PROGRAM Axis05_Auto
VAR
//System_Bit
	Always_ON	:	BOOL	:=TRUE	;//상시 ON 
	Always_OFF	:	BOOL	:=FALSE	;//상시 OFF
END_VAR

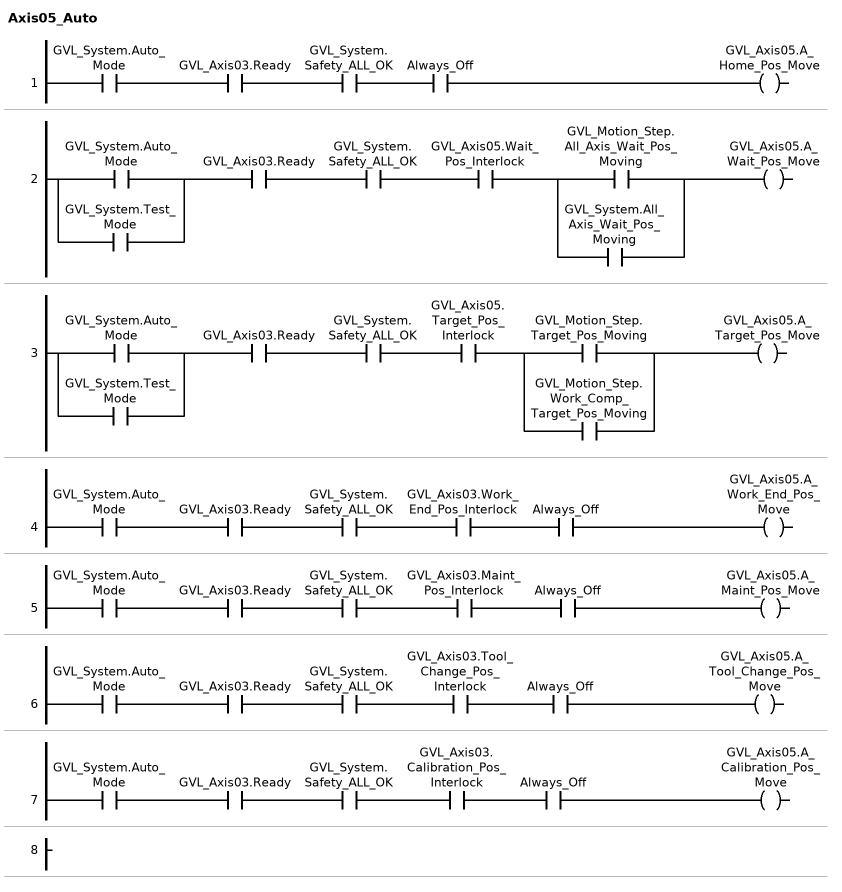
// NETWORK 1
GVL_Axis05.A_Home_Pos_Move := GVL_System.Auto_Mode AND GVL_Axis03.Ready AND GVL_System.Safety_ALL_OK AND Always_Off;

// NETWORK 2
GVL_Axis05.A_Wait_Pos_Move := (GVL_System.Auto_Mode OR GVL_System.Test_Mode) AND GVL_Axis03.Ready AND GVL_System.Safety_ALL_OK AND GVL_Axis05.Wait_Pos_Interlock AND (GVL_Motion_Step.All_Axis_Wait_Pos_Moving OR GVL_System.All_Axis_Wait_Pos_Moving);

// NETWORK 3
GVL_Axis05.A_Target_Pos_Move := (GVL_System.Auto_Mode OR GVL_System.Test_Mode) AND GVL_Axis03.Ready AND GVL_System.Safety_ALL_OK AND GVL_Axis05.Target_Pos_Interlock AND (GVL_Motion_Step.Target_Pos_Moving OR GVL_Motion_Step.Work_Comp_Target_Pos_Moving);

// NETWORK 4
GVL_Axis05.A_Work_End_Pos_Move := GVL_System.Auto_Mode AND GVL_Axis03.Ready AND GVL_System.Safety_ALL_OK AND GVL_Axis03.Work_End_Pos_Interlock AND Always_Off;

// NETWORK 5
GVL_Axis05.A_Maint_Pos_Move := GVL_System.Auto_Mode AND GVL_Axis03.Ready AND GVL_System.Safety_ALL_OK AND GVL_Axis03.Maint_Pos_Interlock AND Always_Off;

// NETWORK 6
GVL_Axis05.A_Tool_Change_Pos_Move := GVL_System.Auto_Mode AND GVL_Axis03.Ready AND GVL_System.Safety_ALL_OK AND GVL_Axis03.Tool_Change_Pos_Interlock AND Always_Off;

// NETWORK 7
GVL_Axis05.A_Calibration_Pos_Move := GVL_System.Auto_Mode AND GVL_Axis03.Ready AND GVL_System.Safety_ALL_OK AND GVL_Axis03.Calibration_Pos_Interlock AND Always_Off;

// NETWORK 8

END_PROGRAM

(* stored: Version 1.1.0.1, ProductVersion 3.1.4024.15
   POU Axis05_Auto: Id {a556c58e-1b45-4a45-ad62-b9b9b34a80ae}, SpecialFunc None *)
